// TwinCAT 3 PLC project ADS_Server
// ProgramVersion: 3.1.4023.0
// libraries:
//   Tc2_Standard, * (Beckhoff Automation GmbH)
//   Tc2_System, * (Beckhoff Automation GmbH)
//   Tc3_Module, * (Beckhoff Automation GmbH)
// project tree:
//   / GlobalTextList.TcGTLO, PlcTask.TcTTO, Visualization Manager.TcVMO (not stored)
//   POUs/ MAIN.TcPOU
//   VISUs/ Visualization.TcVIS

CONFIGURATION ADS_Server
    RESOURCE PLC ON TwinCAT3
        TASK PlcTask(INTERVAL := T#10ms, PRIORITY := 20);
        PROGRAM MAIN WITH PlcTask : MAIN;
    END_RESOURCE
END_CONFIGURATION

// ---- POUs/MAIN.TcPOU
PROGRAM MAIN
VAR
	bRecivedRequest : BOOL; //we recive the request
	bAnswerTheRequest : BOOL; //we decide whether or not we accept the request
	bRequestIndicator : BOOL; //the use of this variable is for indication in the visualization
	rWrittenValue : LREAL; //we get the new value written
	rRequestedValue : LREAL;
	bAccept : BOOL; //button to accept the request
	bDeny : BOOL; //button to deny the request
	iPositionMotor : DINT; //the position of the motor
	bReadPositionButton : BOOL;
	
	iState : UINT;
	
	fbResetRequest : TON;
	fbReadRequestedValue : ADSREAD;
	fbReadPositionValue : ADSREAD; //reading the position of the motor from the master PLC
END_VAR

CASE iState OF
	0: //wait for the request
		IF bRecivedRequest THEN
			iState := 10;
		END_IF
	10: //accept or deny the request
		IF bAccept THEN
			bAnswerTheRequest := TRUE;
			bRecivedRequest := FALSE;
			iState := 20;
		ELSIF bDeny THEN
			bAnswerTheRequest := FALSE;
			bRecivedRequest := FALSE;
			iState := 0;
		END_IF
	20: //the value has been written wait 3s then reset the answer and wait for a new request
		fbResetRequest.IN := TRUE;
		IF fbResetRequest.Q THEN
			bAnswerTheRequest := FALSE;
			fbResetRequest.IN := FALSE;
			iState := 0;
		END_IF	
END_CASE
IF iState = 10 THEN
	bRequestIndicator := TRUE;
ELSE
	bRequestIndicator := FALSE;
END_IF
fbReadRequestedValue(NetId := '10.0.20.83.1.1', //we read the requested value aand display it so the user can decide whether or not he accepts
					 Port := 851,
					 IDXGRP := 16#4040,
					 IDXOFFS := 386880,
					 LEN := SIZEOF(rRequestedValue),
					 DESTADDR := ADR(rRequestedValue),
					 Read := bRequestIndicator);

fbReadPositionValue(NetId := '10.0.20.83.1.1',
					Port := 851,
					IDXGRP := 16#4040,
					IDXOFFS := 386960,
					LEN := SIZEOF(iPositionMotor),
					DESTADDR := ADR(iPositionMotor),
					Read := bReadPositionButton);
					
fbResetRequest(PT := T#3S);

END_PROGRAM

// ---- GlobalTextList.TcGTLO
TEXTLIST GlobalTextList
  771 = 'Accept Request'
  449 = 'Actual value: %f'
  173 = 'Deny Request'
  380 = 'Motor Position: %i'
  217 = 'Requested value: %f'
  919 = 'Value: %f'
END_TEXTLIST

// ---- VISUs/Visualization.TcVIS
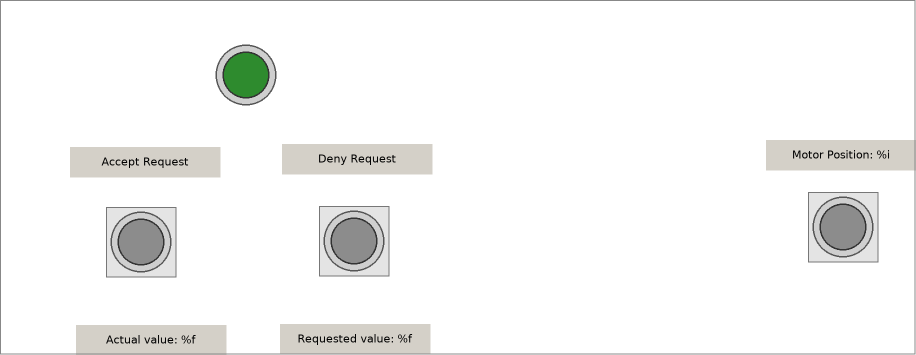
VISUALIZATION Visualization  // 916x355
    PushSwitch (319,206 70x70), variable: MAIN.bDeny, behaviour: TAP, style: Switch-PushSwitch-Gray
    PushSwitch (106,207 70x70), variable: MAIN.bAccept, behaviour: TAP, style: Switch-PushSwitch-Gray
    Textfield (282,144 150x30), "Deny Request"
    Textfield (76,325 150x30), "Actual value: %f", text variable: MAIN.rWrittenValue
    Textfield (70,147 150x30), "Accept Request"
    Textfield (280,324 150x30), "Requested value: %f", text variable: MAIN.rRequestedValue
    Lamp1 (211,40 70x70), variable: MAIN.bRequestIndicator, style: Lamp-Lamp1-Green
    PushSwitch (808,192 70x70), variable: MAIN.bReadPositionButton, behaviour: TAP, style: Switch-PushSwitch-Gray
    Textfield (766,140 150x30), "Motor Position: %i", text variable: MAIN.iPositionMotor
END_VISUALIZATION
